# EPICS IOC start-up script: require/3.1.2/siteMods/iocStats/3.1.16/iocStats.iocsh
# ### IOCSTATS iocsh  ###
#- ###################################################
#- IOCNAME          - IOCSTATS IOCNAME
#- ###################################################

dbLoadRecords("iocAdminSoft-ess.db", "IOC=$(IOCNAME)-IocStats")
